// TIA Portal project "MD_Server_V18" (V18)

(* hardware
DEVICE "S7-1200 station_1"  S7-1200 Station
   slot 0: "Rack_0"  S7-1200 Rack  Rack  V1.0
   slot 1: "PLC_1"  CPU 1215C DC/DC/DC  6ES7 215-1AG40-0XB0  V4.2
   slot 2: "AI 4x13BIT/AQ 2x14BIT_1"  6ES7 234-4HE32-0XB0  V2.0
*)

// ===== PLC "PLC_1"  CPU 1215C DC/DC/DC =====

DATA_BLOCK "MB_data"   // DB1
{ S7_Optimized_Access := 'TRUE' }
VERSION : 0.1
   VAR
      Booleens : Array[0..100] of Bool;
      Data : Array[0..100] of Int;
   END_VAR
BEGIN
END_DATA_BLOCK

DATA_BLOCK "MB_Server_CONFIG"   // DB2
{ S7_Optimized_Access := 'TRUE' }
VERSION : 0.1
   VAR
      MBServer : TCON_IP_v4;
      MB_NDR : Bool;
      MB_DR : Bool;
      MB_ERROR : Bool;
      MB_STATUS : Word;
   END_VAR
BEGIN
   MBServer.InterfaceId := 64;
   MBServer.LocalPort := 502;
   MBServer.ID := 16#01;
END_DATA_BLOCK

ORGANIZATION_BLOCK "Main"   // OB1, LAD, ProgramCycle
TITLE = "Main Program Sweep (Cycle)"
{ S7_Optimized_Access := 'TRUE' }
VERSION : 0.1
   VAR_INPUT
      Initial_Call : Bool;   // Initial call of this OB
      Remanence : Bool;   // =True, if remanent data are available
   END_VAR
BEGIN

REGION Network 1
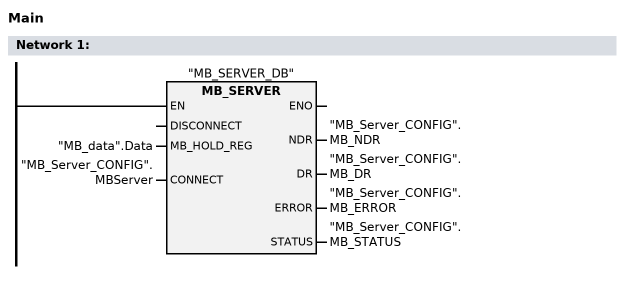
   "MB_SERVER_DB"(MB_HOLD_REG := "MB_data".Data,   // MB_SERVER
                  CONNECT := "MB_Server_CONFIG".MBServer,
                  NDR => "MB_Server_CONFIG".MB_NDR,
                  DR => "MB_Server_CONFIG".MB_DR,
                  ERROR => "MB_Server_CONFIG".MB_ERROR,
                  STATUS => "MB_Server_CONFIG".MB_STATUS);
END_REGION
END_ORGANIZATION_BLOCK